Fanuc KAREL source: ko00093.KL

-- PROVISIONAL review KL for V770-1; original PC SHA256 db503db09578bddb17bab137925ffe60cfdc7f639b9dd03cefd40ad4a982d04d
-- Incomplete behavior may be omitted. Consult companion uncertainty JSON. Do not deploy.
PROGRAM KO00093
%NOLOCKGROUP
BEGIN
  -- UNRESOLVED_PC offsets 5-12; opcodes 9D,23
  -- UNRESOLVED_PC offsets 17-69; opcodes 27,27,49,7E,AD,27,49,7E,AD,22,31,7E,4A
  -- UNRESOLVED_PC offsets 74-78; opcodes 7F
END KO00093
